(* CoDeSys 2.3 export: IP_ADDRESS.EXP *)

(* POU Moje funkcje/IP_ADDRESS, ST *)
FUNCTION IP_ADDRESS : DWORD
VAR_INPUT
	IP_ADR	:	STRING;
END_VAR
VAR
	Address 	:	DWORD;
	Value		:	WORD;
	DecimalPos	:	INT;
	Rest		:	STRING;
END_VAR
Address := STRING_TO_WORD(IP_ADR);
IF (Address <= 255) AND (Address >= 0) THEN
	DecimalPos := FIND(IP_ADR,'.');
	IF DecimalPos <> 0 THEN
		Rest := RIGHT(IP_ADR,LEN(IP_ADR) - DecimalPos);
		Value := STRING_TO_WORD(Rest);
		IF (Value <= 255) AND (Value >= 0) THEN
			Address := (Address * 16#0100) + Value;

			DecimalPos := FIND(Rest,'.');
			IF DecimalPos <> 0 THEN
				Rest := RIGHT(IP_ADR,LEN(Rest) - DecimalPos);
				Value := STRING_TO_WORD(Rest);
				IF (Value <= 255) AND (Value >= 0) THEN
					Address := (Address * 16#0100) + Value;

					DecimalPos := FIND(Rest,'.');
					IF DecimalPos <> 0 THEN
						Rest := RIGHT(IP_ADR,LEN(Rest) - DecimalPos);
						Value := STRING_TO_WORD(Rest);
						IF (Value <= 255) AND (Value >= 0) THEN
							Address := (Address * 16#0100) + Value;
						ELSE
							Address := 0;
						END_IF
					ELSE
						Address := 0;
					END_IF
				ELSE
					Address := 0;
				END_IF
			ELSE
				Address := 0;
			END_IF
		ELSE
			Address := 0;
		END_IF
	ELSE
		Address := 0;
	END_IF
ELSE
	Address := 0;
END_IF
IP_ADDRESS := Address;
END_FUNCTION
